// ---- DUTs/IO/Topology/Beckhoff_EJ5xxx_DF22D5A3.TcDUT
{attribute addProperty BoxType "EK1100-0000-0018"}
{attribute addProperty Id "Beckhoff_EJ5xxxEK1122Beckhoff_EJ5xxxEK1122_0744EC7C162A_0001_EJ5002_0000_0016EJ5002_8228306817822.25A_0002_EJ5002_0000_0017EJ5002_960CC6F117822.25A_0003_EJ5101_0000_0016EJ5101_6012872616220.25A_0004_EJ5151_0000_0016EJ5151_0AC1A36D19424.25"}
{attribute addProperty CRC "3743602083"}
{attribute addProperty SizeInBites "728"}
{attribute addProperty SizeInBytes "91"}
TYPE Beckhoff_EJ5xxx_DF22D5A3 EXTENDS EK1100_179A0949 :
STRUCT
	{attribute addProperty Name "Beckhoff_EJ5xxxEK1122"}
	Beckhoff_EJ5xxxEK1122 : Beckhoff_EJ5xxxEK1122_0744EC7C;
	{attribute addProperty Name "A_0001_EJ5002_0000_0016"}
	A_0001_EJ5002_0000_0016 : EJ5002_82283068;
	{attribute addProperty Name "A_0002_EJ5002_0000_0017"}
	A_0002_EJ5002_0000_0017 : EJ5002_960CC6F1;
	{attribute addProperty Name "A_0003_EJ5101_0000_0016"}
	A_0003_EJ5101_0000_0016 : EJ5101_60128726;
	{attribute addProperty Name "A_0004_EJ5151_0000_0016"}
	A_0004_EJ5151_0000_0016 : EJ5151_0AC1A36D;
END_STRUCT
END_TYPE

// ---- DUTs/IO/Topology/Beckhoff_EJ6xxxEK1122_30779985.TcDUT
{attribute addProperty BoxType "EK1122-0000-0018"}
{attribute addProperty Id "Beckhoff_EJ6xxxsub_EK1100EK1100_179A0949162"}
{attribute addProperty CRC "813144453"}
{attribute addProperty SizeInBites "16"}
{attribute addProperty SizeInBytes "2"}
TYPE Beckhoff_EJ6xxxEK1122_30779985 EXTENDS EK1122_179A0949 :
STRUCT
	{attribute addProperty Name "Beckhoff_EJ6xxxsub_EK1100"}
	Beckhoff_EJ6xxxsub_EK1100 : EK1100_179A0949;
END_STRUCT
END_TYPE

// ---- DUTs/IO/Topology/Beckhoff_EJ6xxx_A0E5C2C0.TcDUT
{attribute addProperty BoxType "EK1100-0000-0018"}
{attribute addProperty Id "Beckhoff_EJ6xxxEK1122Beckhoff_EJ6xxxEK1122_30779985162A_0001_EJ6002_0000_0016EJ6002_880A624E850106.25A_0002_EJ6224_0000_0016EJ6224_3990B4B417822.25A_0003_EJ6224_0090_0016EJ6224_3990B4B417822.25"}
{attribute addProperty CRC "2699412160"}
{attribute addProperty SizeInBites "1222"}
{attribute addProperty SizeInBytes "152.75"}
TYPE Beckhoff_EJ6xxx_A0E5C2C0 EXTENDS EK1100_179A0949 :
STRUCT
	{attribute addProperty Name "Beckhoff_EJ6xxxEK1122"}
	Beckhoff_EJ6xxxEK1122 : Beckhoff_EJ6xxxEK1122_30779985;
	{attribute addProperty Name "A_0001_EJ6002_0000_0016"}
	A_0001_EJ6002_0000_0016 : EJ6002_880A624E;
	{attribute addProperty Name "A_0002_EJ6224_0000_0016"}
	A_0002_EJ6224_0000_0016 : EJ6224_3990B4B4;
	{attribute addProperty Name "A_0003_EJ6224_0090_0016"}
	A_0003_EJ6224_0090_0016 : EJ6224_3990B4B4;
END_STRUCT
END_TYPE

// ---- DUTs/IO/Topology/Beckhoff_EJ7xxxEK1122_22994AD2.TcDUT
{attribute addProperty BoxType "EK1122-0000-0018"}
{attribute addProperty Id "Beckhoff_EJ7xxxsub_EK1100EK1100_179A0949162"}
{attribute addProperty CRC "580471506"}
{attribute addProperty SizeInBites "16"}
{attribute addProperty SizeInBytes "2"}
TYPE Beckhoff_EJ7xxxEK1122_22994AD2 EXTENDS EK1122_179A0949 :
STRUCT
	{attribute addProperty Name "Beckhoff_EJ7xxxsub_EK1100"}
	Beckhoff_EJ7xxxsub_EK1100 : EK1100_179A0949;
END_STRUCT
END_TYPE

// ---- DUTs/IO/Topology/Beckhoff_EJ7xxx_9F75012E.TcDUT
{attribute addProperty BoxType "EK1100-0000-0018"}
{attribute addProperty Id "Beckhoff_EJ7xxxEK1122Beckhoff_EJ7xxxEK1122_22994AD2162A_0001_EJ7031_0000_0026EJ7031_26D8313822628.25A_0002_EJ7037_0000_0020EJ7037_F30AD12822628.25A_0003_EJ7041_0052_0016EJ7041_26D8313822628.25A_0004_EJ7047_0000_0018EJ7047_F30AD12822628.25A_0005_EJ7047_0000_0019EJ7047_F30AD12822628.25A_0006_EJ7047_0000_0020EJ7047_F30AD12822628.25A_0007_EJ7342_0000_0019EJ7342_E03DC37137046.25A_0008_EJ7342_0000_0020EJ7342_E2585B8337046.25A_0009_EJ7211_0010_0026EJ7211_83D4128E25031.25A_0010_EJ7211_0010_0027EJ7211_83D4128E25031.25A_0011_EJ7211_0010_0028EJ7211_83D4128E25031.25A_0012_EJ7211_0010_0029EJ7211_83D4128E25031.25A_0013_EJ7211_0010_0030EJ7211_2D7B43DC25832.25A_0014_EJ7211_0010_0031EJ7211_2D7B43DC25832.25A_0015_EJ7211_0010_0032EJ7211_2D7B43DC25832.25A_0016_EJ7211_0011_0026EJ7211_789C0F5925031.25A_0017_EJ7211_0011_0027EJ7211_789C0F5925031.25A_0018_EJ7211_0011_0028EJ7211_789C0F5925031.25A_0019_EJ7211_0011_0029EJ7211_789C0F5925031.25A_0020_EJ7211_0011_0030EJ7211_789C0F5925031.25A_0021_EJ7211_0011_0031EJ7211_789C0F5925031.25A_0022_EJ7211_0011_0032EJ7211_789C0F5925031.25A_0023_EJ7211_9414_0029EJ7211_83D4128E25031.25A_0024_EJ7211_9414_0030EJ7211_5D87091826633.25A_0025_EJ7211_9414_0031EJ7211_5D87091826633.25A_0026_EJ7211_9414_0032EJ7211_5D87091826633.25A_0027_EJ7211_9415_0029EJ7211_789C0F5925031.25A_0028_EJ7211_9415_0030EJ7211_789C0F5925031.25A_0029_EJ7211_9415_0031EJ7211_789C0F5925031.25A_0030_EJ7211_9415_0032EJ7211_789C0F5925031.25A_0031_EJ7334_0008_0016EJ7334_68079CA927434.25A_0032_EJ7411_0000_0018EJ7411_675FBD0529036.25"}
{attribute addProperty CRC "2675245358"}
{attribute addProperty SizeInBites "8248"}
{attribute addProperty SizeInBytes "1031"}
TYPE Beckhoff_EJ7xxx_9F75012E EXTENDS EK1100_179A0949 :
STRUCT
	{attribute addProperty Name "Beckhoff_EJ7xxxEK1122"}
	Beckhoff_EJ7xxxEK1122 : Beckhoff_EJ7xxxEK1122_22994AD2;
	{attribute addProperty Name "A_0001_EJ7031_0000_0026"}
	A_0001_EJ7031_0000_0026 : EJ7031_26D83138;
	{attribute addProperty Name "A_0002_EJ7037_0000_0020"}
	A_0002_EJ7037_0000_0020 : EJ7037_F30AD128;
	{attribute addProperty Name "A_0003_EJ7041_0052_0016"}
	A_0003_EJ7041_0052_0016 : EJ7041_26D83138;
	{attribute addProperty Name "A_0004_EJ7047_0000_0018"}
	A_0004_EJ7047_0000_0018 : EJ7047_F30AD128;
	{attribute addProperty Name "A_0005_EJ7047_0000_0019"}
	A_0005_EJ7047_0000_0019 : EJ7047_F30AD128;
	{attribute addProperty Name "A_0006_EJ7047_0000_0020"}
	A_0006_EJ7047_0000_0020 : EJ7047_F30AD128;
	{attribute addProperty Name "A_0007_EJ7342_0000_0019"}
	A_0007_EJ7342_0000_0019 : EJ7342_E03DC371;
	{attribute addProperty Name "A_0008_EJ7342_0000_0020"}
	A_0008_EJ7342_0000_0020 : EJ7342_E2585B83;
	{attribute addProperty Name "A_0009_EJ7211_0010_0026"}
	A_0009_EJ7211_0010_0026 : EJ7211_83D4128E;
	{attribute addProperty Name "A_0010_EJ7211_0010_0027"}
	A_0010_EJ7211_0010_0027 : EJ7211_83D4128E;
	{attribute addProperty Name "A_0011_EJ7211_0010_0028"}
	A_0011_EJ7211_0010_0028 : EJ7211_83D4128E;
	{attribute addProperty Name "A_0012_EJ7211_0010_0029"}
	A_0012_EJ7211_0010_0029 : EJ7211_83D4128E;
	{attribute addProperty Name "A_0013_EJ7211_0010_0030"}
	A_0013_EJ7211_0010_0030 : EJ7211_2D7B43DC;
	{attribute addProperty Name "A_0014_EJ7211_0010_0031"}
	A_0014_EJ7211_0010_0031 : EJ7211_2D7B43DC;
	{attribute addProperty Name "A_0015_EJ7211_0010_0032"}
	A_0015_EJ7211_0010_0032 : EJ7211_2D7B43DC;
	{attribute addProperty Name "A_0016_EJ7211_0011_0026"}
	A_0016_EJ7211_0011_0026 : EJ7211_789C0F59;
	{attribute addProperty Name "A_0017_EJ7211_0011_0027"}
	A_0017_EJ7211_0011_0027 : EJ7211_789C0F59;
	{attribute addProperty Name "A_0018_EJ7211_0011_0028"}
	A_0018_EJ7211_0011_0028 : EJ7211_789C0F59;
	{attribute addProperty Name "A_0019_EJ7211_0011_0029"}
	A_0019_EJ7211_0011_0029 : EJ7211_789C0F59;
	{attribute addProperty Name "A_0020_EJ7211_0011_0030"}
	A_0020_EJ7211_0011_0030 : EJ7211_789C0F59;
	{attribute addProperty Name "A_0021_EJ7211_0011_0031"}
	A_0021_EJ7211_0011_0031 : EJ7211_789C0F59;
	{attribute addProperty Name "A_0022_EJ7211_0011_0032"}
	A_0022_EJ7211_0011_0032 : EJ7211_789C0F59;
	{attribute addProperty Name "A_0023_EJ7211_9414_0029"}
	A_0023_EJ7211_9414_0029 : EJ7211_83D4128E;
	{attribute addProperty Name "A_0024_EJ7211_9414_0030"}
	A_0024_EJ7211_9414_0030 : EJ7211_5D870918;
	{attribute addProperty Name "A_0025_EJ7211_9414_0031"}
	A_0025_EJ7211_9414_0031 : EJ7211_5D870918;
	{attribute addProperty Name "A_0026_EJ7211_9414_0032"}
	A_0026_EJ7211_9414_0032 : EJ7211_5D870918;
	{attribute addProperty Name "A_0027_EJ7211_9415_0029"}
	A_0027_EJ7211_9415_0029 : EJ7211_789C0F59;
	{attribute addProperty Name "A_0028_EJ7211_9415_0030"}
	A_0028_EJ7211_9415_0030 : EJ7211_789C0F59;
	{attribute addProperty Name "A_0029_EJ7211_9415_0031"}
	A_0029_EJ7211_9415_0031 : EJ7211_789C0F59;
	{attribute addProperty Name "A_0030_EJ7211_9415_0032"}
	A_0030_EJ7211_9415_0032 : EJ7211_789C0F59;
	{attribute addProperty Name "A_0031_EJ7334_0008_0016"}
	A_0031_EJ7334_0008_0016 : EJ7334_68079CA9;
	{attribute addProperty Name "A_0032_EJ7411_0000_0018"}
	A_0032_EJ7411_0000_0018 : EJ7411_675FBD05;
END_STRUCT
END_TYPE

// ---- DUTs/IO/Topology/Beckhoff_EJ9xxxEK1122_DB893B98.TcDUT
{attribute addProperty BoxType "EK1122-0000-0018"}
{attribute addProperty Id "Beckhoff_EJ9xxxsub_EK1100EK1100_179A0949162"}
{attribute addProperty CRC "3683203992"}
{attribute addProperty SizeInBites "16"}
{attribute addProperty SizeInBytes "2"}
TYPE Beckhoff_EJ9xxxEK1122_DB893B98 EXTENDS EK1122_179A0949 :
STRUCT
	{attribute addProperty Name "Beckhoff_EJ9xxxsub_EK1100"}
	Beckhoff_EJ9xxxsub_EK1100 : EK1100_179A0949;
END_STRUCT
END_TYPE

// ---- DUTs/IO/Topology/Beckhoff_EJ9xxx_660B2C8D.TcDUT
{attribute addProperty BoxType "EK1100-0000-0018"}
{attribute addProperty Id "Beckhoff_EJ9xxxEK1122Beckhoff_EJ9xxxEK1122_DB893B98162A_0001_EJ9001_0000_0016EJ9001_179A0949162A_0002_EJ9505_0000_0016EJ9505_13AAEB7E344.25A_0003_EJ9576_0000_0018EJ9576_30D5723B21026.25A_0004_EJ9576_0000_0019EJ9576_8602C5C421827.25A_0005_EJ9576_0000_0020EJ9576_EB67CEB421026.25A_0006_EJ9576_0000_0022EJ9576_EEF1625221827.25"}
{attribute addProperty CRC "1712008333"}
{attribute addProperty SizeInBites "922"}
{attribute addProperty SizeInBytes "115.25"}
TYPE Beckhoff_EJ9xxx_660B2C8D EXTENDS EK1100_179A0949 :
STRUCT
	{attribute addProperty Name "Beckhoff_EJ9xxxEK1122"}
	Beckhoff_EJ9xxxEK1122 : Beckhoff_EJ9xxxEK1122_DB893B98;
	{attribute addProperty Name "A_0001_EJ9001_0000_0016"}
	A_0001_EJ9001_0000_0016 : EJ9001_179A0949;
	{attribute addProperty Name "A_0002_EJ9505_0000_0016"}
	A_0002_EJ9505_0000_0016 : EJ9505_13AAEB7E;
	{attribute addProperty Name "A_0003_EJ9576_0000_0018"}
	A_0003_EJ9576_0000_0018 : EJ9576_30D5723B;
	{attribute addProperty Name "A_0004_EJ9576_0000_0019"}
	A_0004_EJ9576_0000_0019 : EJ9576_8602C5C4;
	{attribute addProperty Name "A_0005_EJ9576_0000_0020"}
	A_0005_EJ9576_0000_0020 : EJ9576_EB67CEB4;
	{attribute addProperty Name "A_0006_EJ9576_0000_0022"}
	A_0006_EJ9576_0000_0022 : EJ9576_EEF16252;
END_STRUCT
END_TYPE

// ---- DUTs/IO/Topology/Beckhoff_EJx9xxEK1122_05D2B413.TcDUT
{attribute addProperty BoxType "EK1122-0000-0018"}
{attribute addProperty Id "Beckhoff_EJx9xxsub_EK1100EK1100_179A0949162"}
{attribute addProperty CRC "97694739"}
{attribute addProperty SizeInBites "16"}
{attribute addProperty SizeInBytes "2"}
TYPE Beckhoff_EJx9xxEK1122_05D2B413 EXTENDS EK1122_179A0949 :
STRUCT
	{attribute addProperty Name "Beckhoff_EJx9xxsub_EK1100"}
	Beckhoff_EJx9xxsub_EK1100 : EK1100_179A0949;
END_STRUCT
END_TYPE

// ---- DUTs/IO/Topology/Beckhoff_EJx9xx_A9128509.TcDUT
{attribute addProperty BoxType "EK1100-0000-0018"}
{attribute addProperty Id "Beckhoff_EJx9xxEK1122Beckhoff_EJx9xxEK1122_05D2B413162A_0001_EJ1914_0000_0017EJ1914_5EB96E2D21026.25A_0002_EJ1914_0000_0018EJ1914_5EB96E2D21026.25A_0003_EJ1918_0000_0017EJ1918_151E5A8221827.25A_0004_EJ1918_0000_0018EJ1918_151E5A8221827.25A_0005_EJ1957_0000_0017EJ1957_6B6926D126032.5A_0006_EJ1957_0000_0018EJ1957_6B6926D126032.5A_0007_EJ2914_0000_0017EJ2914_46D107EB24430.5A_0008_EJ2914_0000_0018EJ2914_46D107EB24430.5A_0009_EJ2918_0000_0017EJ2918_AA36864B28435.5A_0010_EJ2918_0000_0018EJ2918_AA36864B28435.5A_0011_EJ6910_0000_0018EJ6910_4EA245C69812.25A_0012_EJ6910_0000_0020EJ6910_4EA245C69812.25"}
{attribute addProperty CRC "2836563209"}
{attribute addProperty SizeInBites "2644"}
{attribute addProperty SizeInBytes "330.5"}
TYPE Beckhoff_EJx9xx_A9128509 EXTENDS EK1100_179A0949 :
STRUCT
	{attribute addProperty Name "Beckhoff_EJx9xxEK1122"}
	Beckhoff_EJx9xxEK1122 : Beckhoff_EJx9xxEK1122_05D2B413;
	{attribute addProperty Name "A_0001_EJ1914_0000_0017"}
	A_0001_EJ1914_0000_0017 : EJ1914_5EB96E2D;
	{attribute addProperty Name "A_0002_EJ1914_0000_0018"}
	A_0002_EJ1914_0000_0018 : EJ1914_5EB96E2D;
	{attribute addProperty Name "A_0003_EJ1918_0000_0017"}
	A_0003_EJ1918_0000_0017 : EJ1918_151E5A82;
	{attribute addProperty Name "A_0004_EJ1918_0000_0018"}
	A_0004_EJ1918_0000_0018 : EJ1918_151E5A82;
	{attribute addProperty Name "A_0005_EJ1957_0000_0017"}
	A_0005_EJ1957_0000_0017 : EJ1957_6B6926D1;
	{attribute addProperty Name "A_0006_EJ1957_0000_0018"}
	A_0006_EJ1957_0000_0018 : EJ1957_6B6926D1;
	{attribute addProperty Name "A_0007_EJ2914_0000_0017"}
	A_0007_EJ2914_0000_0017 : EJ2914_46D107EB;
	{attribute addProperty Name "A_0008_EJ2914_0000_0018"}
	A_0008_EJ2914_0000_0018 : EJ2914_46D107EB;
	{attribute addProperty Name "A_0009_EJ2918_0000_0017"}
	A_0009_EJ2918_0000_0017 : EJ2918_AA36864B;
	{attribute addProperty Name "A_0010_EJ2918_0000_0018"}
	A_0010_EJ2918_0000_0018 : EJ2918_AA36864B;
	{attribute addProperty Name "A_0011_EJ6910_0000_0018"}
	A_0011_EJ6910_0000_0018 : EJ6910_4EA245C6;
	{attribute addProperty Name "A_0012_EJ6910_0000_0020"}
	A_0012_EJ6910_0000_0020 : EJ6910_4EA245C6;
END_STRUCT
END_TYPE

// ---- DUTs/IO/Topology/EtherCAT_Master_EJxxxx_24234FDA.TcDUT
{attribute addProperty BoxType "IODEVICETYPE_ETHERCATPROT"}
{attribute addProperty Id "Beckhoff_EJ1xxxBeckhoff_EJ1xxx_BA4DEDCC877109.625Beckhoff_EJ2xxxBeckhoff_EJ2xxx_42F4B05B1708213.5Beckhoff_EJ3xxxBeckhoff_EJ3xxx_F355313D4934616.75Beckhoff_EJ4xxxBeckhoff_EJ4xxx_B433EAC71353169.125Beckhoff_EJ5xxxBeckhoff_EJ5xxx_DF22D5A372891Beckhoff_EJ6xxxBeckhoff_EJ6xxx_A0E5C2C01222152.75Beckhoff_EJ7xxxBeckhoff_EJ7xxx_9F75012E82481031Beckhoff_EJ9xxxBeckhoff_EJ9xxx_660B2C8D922115.25Beckhoff_EJx9xxBeckhoff_EJx9xx_A91285092644330.5SyncUnitsSyncUnits_BBFB8ED413016.25InputsInputs_C3133F881088136OutputsOutputs_BAAAC74672090InfoDataInfoData_E9F65A829612"}
{attribute addProperty CRC "606293978"}
{attribute addProperty SizeInBites "24670"}
{attribute addProperty SizeInBytes "3083.75"}
TYPE EtherCAT_Master_EJxxxx_24234FDA :
STRUCT
	{attribute addProperty Name "Beckhoff_EJ1xxx"}
	Beckhoff_EJ1xxx : Beckhoff_EJ1xxx_BA4DEDCC;
	{attribute addProperty Name "Beckhoff_EJ2xxx"}
	Beckhoff_EJ2xxx : Beckhoff_EJ2xxx_42F4B05B;
	{attribute addProperty Name "Beckhoff_EJ3xxx"}
	Beckhoff_EJ3xxx : Beckhoff_EJ3xxx_F355313D;
	{attribute addProperty Name "Beckhoff_EJ4xxx"}
	Beckhoff_EJ4xxx : Beckhoff_EJ4xxx_B433EAC7;
	{attribute addProperty Name "Beckhoff_EJ5xxx"}
	Beckhoff_EJ5xxx : Beckhoff_EJ5xxx_DF22D5A3;
	{attribute addProperty Name "Beckhoff_EJ6xxx"}
	Beckhoff_EJ6xxx : Beckhoff_EJ6xxx_A0E5C2C0;
	{attribute addProperty Name "Beckhoff_EJ7xxx"}
	Beckhoff_EJ7xxx : Beckhoff_EJ7xxx_9F75012E;
	{attribute addProperty Name "Beckhoff_EJ9xxx"}
	Beckhoff_EJ9xxx : Beckhoff_EJ9xxx_660B2C8D;
	{attribute addProperty Name "Beckhoff_EJx9xx"}
	Beckhoff_EJx9xx : Beckhoff_EJx9xx_A9128509;
	{attribute addProperty Name "SyncUnits"}
	SyncUnits : SyncUnits_BBFB8ED4;
	{attribute addProperty Name "Inputs"}
	Inputs : Inputs_C3133F88;
	{attribute addProperty Name "Outputs"}
	Outputs : Outputs_BAAAC746;
	{attribute addProperty Name "InfoData"}
	InfoData : InfoData_E9F65A82;
END_STRUCT
END_TYPE

// ---- DUTs/IO/Topology/Beckhoff_EK11xxEK1122_0F9A1885.TcDUT
{attribute addProperty BoxType "EK1122-0000-0018"}
{attribute addProperty Id "Beckhoff_EK11xxsub_EK1100EK1100_179A0949162A_0001_EK1100_0000_0000EK1100_179A0949162A_0002_EK1100_0000_0001EK1100_179A0949162A_0003_EK1100_0000_0016EK1100_179A0949162A_0004_EK1100_0000_0017EK1100_179A0949162A_0005_EK1100_0000_0018EK1100_179A0949162A_0006_EK1100_0008_0016EK1100_179A0949162A_0009_EK1101_0000_0016EK1101_963BF4D7344.25A_0010_EK1101_0000_0017EK1101_963BF4D7344.25A_0011_EK1101_0000_0018EK1101_963BF4D7344.25A_0012_EK1101_0008_0016EK1101_963BF4D7344.25A_0013_EK1101_0010_0016EK1101_963BF4D7344.25A_0008_EK1100_0030_0017EK1100_179A0949162A_0007_EK1100_0030_0016EK1100_179A0949162"}
{attribute addProperty CRC "261757061"}
{attribute addProperty SizeInBites "314"}
{attribute addProperty SizeInBytes "39.25"}
TYPE Beckhoff_EK11xxEK1122_0F9A1885 EXTENDS EK1122_179A0949 :
STRUCT
	{attribute addProperty Name "Beckhoff_EK11xxsub_EK1100"}
	Beckhoff_EK11xxsub_EK1100 : EK1100_179A0949;
	{attribute addProperty Name "A_0001_EK1100_0000_0000"}
	A_0001_EK1100_0000_0000 : EK1100_179A0949;
	{attribute addProperty Name "A_0002_EK1100_0000_0001"}
	A_0002_EK1100_0000_0001 : EK1100_179A0949;
	{attribute addProperty Name "A_0003_EK1100_0000_0016"}
	A_0003_EK1100_0000_0016 : EK1100_179A0949;
	{attribute addProperty Name "A_0004_EK1100_0000_0017"}
	A_0004_EK1100_0000_0017 : EK1100_179A0949;
	{attribute addProperty Name "A_0005_EK1100_0000_0018"}
	A_0005_EK1100_0000_0018 : EK1100_179A0949;
	{attribute addProperty Name "A_0006_EK1100_0008_0016"}
	A_0006_EK1100_0008_0016 : EK1100_179A0949;
	{attribute addProperty Name "A_0009_EK1101_0000_0016"}
	A_0009_EK1101_0000_0016 : EK1101_963BF4D7;
	{attribute addProperty Name "A_0010_EK1101_0000_0017"}
	A_0010_EK1101_0000_0017 : EK1101_963BF4D7;
	{attribute addProperty Name "A_0011_EK1101_0000_0018"}
	A_0011_EK1101_0000_0018 : EK1101_963BF4D7;
	{attribute addProperty Name "A_0012_EK1101_0008_0016"}
	A_0012_EK1101_0008_0016 : EK1101_963BF4D7;
	{attribute addProperty Name "A_0013_EK1101_0010_0016"}
	A_0013_EK1101_0010_0016 : EK1101_963BF4D7;
	{attribute addProperty Name "A_0008_EK1100_0030_0017"}
	A_0008_EK1100_0030_0017 : EK1100_179A0949;
	{attribute addProperty Name "A_0007_EK1100_0030_0016"}
	A_0007_EK1100_0030_0016 : EK1100_179A0949;
END_STRUCT
END_TYPE

// ---- DUTs/IO/Topology/Beckhoff_EK11xx_C12453FF.TcDUT
{attribute addProperty BoxType "EK1100-0000-0018"}
{attribute addProperty Id "Beckhoff_EK11xxEK1122Beckhoff_EK11xxEK1122_0F9A188531439.25A_0018_EK1110_0043_0016EK1110_179A0949162A_0024_EK1122_0008_0016EK1122_179A0949162A_0023_EK1122_0000_0018EK1122_179A0949162A_0022_EK1122_0000_0017EK1122_179A0949162A_0021_EK1122_0000_0016EK1122_179A0949162A_0020_EK1121_0010_0016EK1121_179A0949162A_0019_EK1110_0044_0016EK1110_179A0949162A_0017_EK1110_0008_0016EK1110_179A0949162A_0016_EK1110_0000_0017EK1110_179A0949162A_0015_EK1110_0000_0016EK1110_179A0949162A_0014_EK1110_0000_0000EK1110_179A0949162"}
{attribute addProperty CRC "3240383487"}
{attribute addProperty SizeInBites "490"}
{attribute addProperty SizeInBytes "61.25"}
TYPE Beckhoff_EK11xx_C12453FF EXTENDS EK1100_179A0949 :
STRUCT
	{attribute addProperty Name "Beckhoff_EK11xxEK1122"}
	Beckhoff_EK11xxEK1122 : Beckhoff_EK11xxEK1122_0F9A1885;
	{attribute addProperty Name "A_0018_EK1110_0043_0016"}
	A_0018_EK1110_0043_0016 : EK1110_179A0949;
	{attribute addProperty Name "A_0024_EK1122_0008_0016"}
	A_0024_EK1122_0008_0016 : EK1122_179A0949;
	{attribute addProperty Name "A_0023_EK1122_0000_0018"}
	A_0023_EK1122_0000_0018 : EK1122_179A0949;
	{attribute addProperty Name "A_0022_EK1122_0000_0017"}
	A_0022_EK1122_0000_0017 : EK1122_179A0949;
	{attribute addProperty Name "A_0021_EK1122_0000_0016"}
	A_0021_EK1122_0000_0016 : EK1122_179A0949;
	{attribute addProperty Name "A_0020_EK1121_0010_0016"}
	A_0020_EK1121_0010_0016 : EK1121_179A0949;
	{attribute addProperty Name "A_0019_EK1110_0044_0016"}
	A_0019_EK1110_0044_0016 : EK1110_179A0949;
	{attribute addProperty Name "A_0017_EK1110_0008_0016"}
	A_0017_EK1110_0008_0016 : EK1110_179A0949;
	{attribute addProperty Name "A_0016_EK1110_0000_0017"}
	A_0016_EK1110_0000_0017 : EK1110_179A0949;
	{attribute addProperty Name "A_0015_EK1110_0000_0016"}
	A_0015_EK1110_0000_0016 : EK1110_179A0949;
	{attribute addProperty Name "A_0014_EK1110_0000_0000"}
	A_0014_EK1110_0000_0000 : EK1110_179A0949;
END_STRUCT
END_TYPE

// ---- DUTs/IO/Topology/Beckhoff_EK12xxEK1122_E9998301.TcDUT
{attribute addProperty BoxType "EK1122-0000-0018"}
{attribute addProperty Id "Beckhoff_EK12xxsub_EK1100EK1100_179A0949162"}
{attribute addProperty CRC "3919151873"}
{attribute addProperty SizeInBites "16"}
{attribute addProperty SizeInBytes "2"}
TYPE Beckhoff_EK12xxEK1122_E9998301 EXTENDS EK1122_179A0949 :
STRUCT
	{attribute addProperty Name "Beckhoff_EK12xxsub_EK1100"}
	Beckhoff_EK12xxsub_EK1100 : EK1100_179A0949;
END_STRUCT
END_TYPE

// ---- DUTs/IO/Topology/Beckhoff_EK12xx_26FD3E4A.TcDUT
{attribute addProperty BoxType "EK1100-0000-0018"}
{attribute addProperty Id "Beckhoff_EK12xxEK1122Beckhoff_EK12xxEK1122_E9998301162"}
{attribute addProperty CRC "654130762"}
{attribute addProperty SizeInBites "16"}
{attribute addProperty SizeInBytes "2"}
TYPE Beckhoff_EK12xx_26FD3E4A EXTENDS EK1100_179A0949 :
STRUCT
	{attribute addProperty Name "Beckhoff_EK12xxEK1122"}
	Beckhoff_EK12xxEK1122 : Beckhoff_EK12xxEK1122_E9998301;
END_STRUCT
END_TYPE

// ---- DUTs/IO/Topology/Beckhoff_EK13xxEK1122_7883D180.TcDUT
{attribute addProperty BoxType "EK1122-0000-0018"}
{attribute addProperty Id "Beckhoff_EK13xxsub_EK1100EK1100_179A0949162A_0001_EK1300_0000_0017EK1300_0EEAC8F2344.25"}
{attribute addProperty CRC "2021904768"}
{attribute addProperty SizeInBites "50"}
{attribute addProperty SizeInBytes "6.25"}
TYPE Beckhoff_EK13xxEK1122_7883D180 EXTENDS EK1122_179A0949 :
STRUCT
	{attribute addProperty Name "Beckhoff_EK13xxsub_EK1100"}
	Beckhoff_EK13xxsub_EK1100 : EK1100_179A0949;
	{attribute addProperty Name "A_0001_EK1300_0000_0017"}
	A_0001_EK1300_0000_0017 : EK1300_0EEAC8F2;
END_STRUCT
END_TYPE

// ---- DUTs/IO/Topology/Beckhoff_EK13xx_F78FC0F8.TcDUT
{attribute addProperty BoxType "EK1100-0000-0018"}
{attribute addProperty Id "Beckhoff_EK13xxEK1122Beckhoff_EK13xxEK1122_7883D180506.25A_0003_EK1322_0000_0017EK1322_0EEAC8F2344.25A_0002_EK1310_0000_0017EK1310_0EEAC8F2344.25"}
{attribute addProperty CRC "4153393400"}
{attribute addProperty SizeInBites "118"}
{attribute addProperty SizeInBytes "14.75"}
TYPE Beckhoff_EK13xx_F78FC0F8 EXTENDS EK1100_179A0949 :
STRUCT
	{attribute addProperty Name "Beckhoff_EK13xxEK1122"}
	Beckhoff_EK13xxEK1122 : Beckhoff_EK13xxEK1122_7883D180;
	{attribute addProperty Name "A_0003_EK1322_0000_0017"}
	A_0003_EK1322_0000_0017 : EK1322_0EEAC8F2;
	{attribute addProperty Name "A_0002_EK1310_0000_0017"}
	A_0002_EK1310_0000_0017 : EK1310_0EEAC8F2;
END_STRUCT
END_TYPE

// ---- DUTs/IO/Topology/Beckhoff_EK15xxEK1122_F4825052.TcDUT
{attribute addProperty BoxType "EK1122-0000-0018"}
{attribute addProperty Id "Beckhoff_EK15xxsub_EK1100EK1100_179A0949162A_0001_EK1501_0000_0016EK1501_963BF4D7344.25A_0002_EK1501_0000_0017EK1501_963BF4D7344.25A_0003_EK1501_0000_0018EK1501_963BF4D7344.25A_0004_EK1501_0000_0019EK1501_963BF4D7344.25A_0005_EK1501_0010_0016EK1501_963BF4D7344.25A_0006_EK1501_0010_0017EK1501_963BF4D7344.25A_0007_EK1501_0010_0018EK1501_963BF4D7344.25A_0008_EK1501_0100_0016EK1501_963BF4D7344.25A_0020_EK1541_0000_0016EK1541_963BF4D7344.25A_0021_EK1541_0000_0017EK1541_963BF4D7344.25A_0022_EK1541_0000_0018EK1541_963BF4D7344.25"}
{attribute addProperty CRC "4102180946"}
{attribute addProperty SizeInBites "390"}
{attribute addProperty SizeInBytes "48.75"}
TYPE Beckhoff_EK15xxEK1122_F4825052 EXTENDS EK1122_179A0949 :
STRUCT
	{attribute addProperty Name "Beckhoff_EK15xxsub_EK1100"}
	Beckhoff_EK15xxsub_EK1100 : EK1100_179A0949;
	{attribute addProperty Name "A_0001_EK1501_0000_0016"}
	A_0001_EK1501_0000_0016 : EK1501_963BF4D7;
	{attribute addProperty Name "A_0002_EK1501_0000_0017"}
	A_0002_EK1501_0000_0017 : EK1501_963BF4D7;
	{attribute addProperty Name "A_0003_EK1501_0000_0018"}
	A_0003_EK1501_0000_0018 : EK1501_963BF4D7;
	{attribute addProperty Name "A_0004_EK1501_0000_0019"}
	A_0004_EK1501_0000_0019 : EK1501_963BF4D7;
	{attribute addProperty Name "A_0005_EK1501_0010_0016"}
	A_0005_EK1501_0010_0016 : EK1501_963BF4D7;
	{attribute addProperty Name "A_0006_EK1501_0010_0017"}
	A_0006_EK1501_0010_0017 : EK1501_963BF4D7;
	{attribute addProperty Name "A_0007_EK1501_0010_0018"}
	A_0007_EK1501_0010_0018 : EK1501_963BF4D7;
	{attribute addProperty Name "A_0008_EK1501_0100_0016"}
	A_0008_EK1501_0100_0016 : EK1501_963BF4D7;
	{attribute addProperty Name "A_0020_EK1541_0000_0016"}
	A_0020_EK1541_0000_0016 : EK1541_963BF4D7;
	{attribute addProperty Name "A_0021_EK1541_0000_0017"}
	A_0021_EK1541_0000_0017 : EK1541_963BF4D7;
	{attribute addProperty Name "A_0022_EK1541_0000_0018"}
	A_0022_EK1541_0000_0018 : EK1541_963BF4D7;
END_STRUCT
END_TYPE

// ---- DUTs/IO/Topology/Beckhoff_EK15xx_2CCE234B.TcDUT
{attribute addProperty BoxType "EK1100-0000-0018"}
{attribute addProperty Id "Beckhoff_EK15xxEK1122Beckhoff_EK15xxEK1122_F482505239048.75A_0025_EK1561_0000_0018EK1561_179A0949162A_0024_EK1561_0000_0017EK1561_179A0949162A_0023_EK1561_0000_0016EK1561_179A0949162A_0019_EK1521_0010_0020EK1521_179A0949162A_0018_EK1521_0010_0019EK1521_179A0949162A_0017_EK1521_0010_0018EK1521_179A0949162A_0016_EK1521_0010_0017EK1521_179A0949162A_0015_EK1521_0010_0016EK1521_179A0949162A_0014_EK1521_0000_0021EK1521_179A0949162A_0013_EK1521_0000_0020EK1521_179A0949162A_0012_EK1521_0000_0019EK1521_179A0949162A_0011_EK1521_0000_0018EK1521_179A0949162A_0010_EK1521_0000_0017EK1521_179A0949162A_0009_EK1521_0000_0016EK1521_179A0949162"}
{attribute addProperty CRC "751706955"}
{attribute addProperty SizeInBites "614"}
{attribute addProperty SizeInBytes "76.75"}
TYPE Beckhoff_EK15xx_2CCE234B EXTENDS EK1100_179A0949 :
STRUCT
	{attribute addProperty Name "Beckhoff_EK15xxEK1122"}
	Beckhoff_EK15xxEK1122 : Beckhoff_EK15xxEK1122_F4825052;
	{attribute addProperty Name "A_0025_EK1561_0000_0018"}
	A_0025_EK1561_0000_0018 : EK1561_179A0949;
	{attribute addProperty Name "A_0024_EK1561_0000_0017"}
	A_0024_EK1561_0000_0017 : EK1561_179A0949;
	{attribute addProperty Name "A_0023_EK1561_0000_0016"}
	A_0023_EK1561_0000_0016 : EK1561_179A0949;
	{attribute addProperty Name "A_0019_EK1521_0010_0020"}
	A_0019_EK1521_0010_0020 : EK1521_179A0949;
	{attribute addProperty Name "A_0018_EK1521_0010_0019"}
	A_0018_EK1521_0010_0019 : EK1521_179A0949;
	{attribute addProperty Name "A_0017_EK1521_0010_0018"}
	A_0017_EK1521_0010_0018 : EK1521_179A0949;
	{attribute addProperty Name "A_0016_EK1521_0010_0017"}
	A_0016_EK1521_0010_0017 : EK1521_179A0949;
	{attribute addProperty Name "A_0015_EK1521_0010_0016"}
	A_0015_EK1521_0010_0016 : EK1521_179A0949;
	{attribute addProperty Name "A_0014_EK1521_0000_0021"}
	A_0014_EK1521_0000_0021 : EK1521_179A0949;
	{attribute addProperty Name "A_0013_EK1521_0000_0020"}
	A_0013_EK1521_0000_0020 : EK1521_179A0949;
	{attribute addProperty Name "A_0012_EK1521_0000_0019"}
	A_0012_EK1521_0000_0019 : EK1521_179A0949;
	{attribute addProperty Name "A_0011_EK1521_0000_0018"}
	A_0011_EK1521_0000_0018 : EK1521_179A0949;
	{attribute addProperty Name "A_0010_EK1521_0000_0017"}
	A_0010_EK1521_0000_0017 : EK1521_179A0949;
	{attribute addProperty Name "A_0009_EK1521_0000_0016"}
	A_0009_EK1521_0000_0016 : EK1521_179A0949;
END_STRUCT
END_TYPE

// ---- DUTs/IO/Topology/Beckhoff_EK18xxEK1122_46BB19D8.TcDUT
{attribute addProperty BoxType "EK1122-0000-0018"}
{attribute addProperty Id "Beckhoff_EK18xxsub_EK1100EK1100_179A0949162A_0001_EK1814_0000_0016EK1814_97B4DD118210.25A_0002_EK1814_0000_0017EK1814_97B4DD118210.25A_0003_EK1814_0000_0018EK1814_97B4DD118210.25A_0004_EK1814_0000_0019EK1814_97B4DD118210.25A_0005_EK1818_0000_0016EK1818_5F755A8411414.25A_0006_EK1818_0000_0017EK1818_5F755A8411414.25A_0007_EK1818_0000_0018EK1818_5F755A8411414.25A_0008_EK1828_0000_0016EK1828_A5978B6311414.25A_0009_EK1828_0000_0017EK1828_A5978B6311414.25A_0010_EK1828_0000_0018EK1828_A5978B6311414.25A_0011_EK1828_0010_0016EK1828_A854BE6D8110.125A_0012_EK1828_0010_0017EK1828_A854BE6D8110.125A_0013_EK1828_0010_0018EK1828_A854BE6D8110.125"}
{attribute addProperty CRC "1186666968"}
{attribute addProperty SizeInBites "1271"}
{attribute addProperty SizeInBytes "158.875"}
TYPE Beckhoff_EK18xxEK1122_46BB19D8 EXTENDS EK1122_179A0949 :
STRUCT
	{attribute addProperty Name "Beckhoff_EK18xxsub_EK1100"}
	Beckhoff_EK18xxsub_EK1100 : EK1100_179A0949;
	{attribute addProperty Name "A_0001_EK1814_0000_0016"}
	A_0001_EK1814_0000_0016 : EK1814_97B4DD11;
	{attribute addProperty Name "A_0002_EK1814_0000_0017"}
	A_0002_EK1814_0000_0017 : EK1814_97B4DD11;
	{attribute addProperty Name "A_0003_EK1814_0000_0018"}
	A_0003_EK1814_0000_0018 : EK1814_97B4DD11;
	{attribute addProperty Name "A_0004_EK1814_0000_0019"}
	A_0004_EK1814_0000_0019 : EK1814_97B4DD11;
	{attribute addProperty Name "A_0005_EK1818_0000_0016"}
	A_0005_EK1818_0000_0016 : EK1818_5F755A84;
	{attribute addProperty Name "A_0006_EK1818_0000_0017"}
	A_0006_EK1818_0000_0017 : EK1818_5F755A84;
	{attribute addProperty Name "A_0007_EK1818_0000_0018"}
	A_0007_EK1818_0000_0018 : EK1818_5F755A84;
	{attribute addProperty Name "A_0008_EK1828_0000_0016"}
	A_0008_EK1828_0000_0016 : EK1828_A5978B63;
	{attribute addProperty Name "A_0009_EK1828_0000_0017"}
	A_0009_EK1828_0000_0017 : EK1828_A5978B63;
	{attribute addProperty Name "A_0010_EK1828_0000_0018"}
	A_0010_EK1828_0000_0018 : EK1828_A5978B63;
	{attribute addProperty Name "A_0011_EK1828_0010_0016"}
	A_0011_EK1828_0010_0016 : EK1828_A854BE6D;
	{attribute addProperty Name "A_0012_EK1828_0010_0017"}
	A_0012_EK1828_0010_0017 : EK1828_A854BE6D;
	{attribute addProperty Name "A_0013_EK1828_0010_0018"}
	A_0013_EK1828_0010_0018 : EK1828_A854BE6D;
END_STRUCT
END_TYPE

// ---- DUTs/IO/Topology/Beckhoff_EK18xx_2BB31392.TcDUT
{attribute addProperty BoxType "EK1100-0000-0018"}
{attribute addProperty Id "Beckhoff_EK18xxEK1122Beckhoff_EK18xxEK1122_46BB19D81271158.875"}
{attribute addProperty CRC "733156242"}
{attribute addProperty SizeInBites "1271"}
{attribute addProperty SizeInBytes "158.875"}
TYPE Beckhoff_EK18xx_2BB31392 EXTENDS EK1100_179A0949 :
STRUCT
	{attribute addProperty Name "Beckhoff_EK18xxEK1122"}
	Beckhoff_EK18xxEK1122 : Beckhoff_EK18xxEK1122_46BB19D8;
END_STRUCT
END_TYPE

// ---- DUTs/IO/Topology/Beckhoff_EKM1xxxEK1122_7DC4CCD1.TcDUT
{attribute addProperty BoxType "EK1122-0000-0018"}
{attribute addProperty Id "Beckhoff_EKM1xxxsub_EK1100EK1100_179A0949162A_0001_EKM1101_0000_0016EKM1101_87969BFD51464.25A_0002_EKM1101_0000_0017EKM1101_87969BFD51464.25A_0003_EKM1101_0000_0018EKM1101_87969BFD51464.25A_0004_EKM1101_0000_0019EKM1101_87969BFD51464.25A_0005_EKM1101_0000_0020EKM1101_87969BFD51464.25"}
{attribute addProperty CRC "2110049489"}
{attribute addProperty SizeInBites "2586"}
{attribute addProperty SizeInBytes "323.25"}
TYPE Beckhoff_EKM1xxxEK1122_7DC4CCD1 EXTENDS EK1122_179A0949 :
STRUCT
	{attribute addProperty Name "Beckhoff_EKM1xxxsub_EK1100"}
	Beckhoff_EKM1xxxsub_EK1100 : EK1100_179A0949;
	{attribute addProperty Name "A_0001_EKM1101_0000_0016"}
	A_0001_EKM1101_0000_0016 : EKM1101_87969BFD;
	{attribute addProperty Name "A_0002_EKM1101_0000_0017"}
	A_0002_EKM1101_0000_0017 : EKM1101_87969BFD;
	{attribute addProperty Name "A_0003_EKM1101_0000_0018"}
	A_0003_EKM1101_0000_0018 : EKM1101_87969BFD;
	{attribute addProperty Name "A_0004_EKM1101_0000_0019"}
	A_0004_EKM1101_0000_0019 : EKM1101_87969BFD;
	{attribute addProperty Name "A_0005_EKM1101_0000_0020"}
	A_0005_EKM1101_0000_0020 : EKM1101_87969BFD;
END_STRUCT
END_TYPE

// ---- DUTs/IO/Topology/Beckhoff_EKM1xxx_A6D53207.TcDUT
{attribute addProperty BoxType "EK1100-0000-0018"}
{attribute addProperty Id "Beckhoff_EKM1xxxEK1122Beckhoff_EKM1xxxEK1122_7DC4CCD12586323.25"}
{attribute addProperty CRC "2798989831"}
{attribute addProperty SizeInBites "2586"}
{attribute addProperty SizeInBytes "323.25"}
TYPE Beckhoff_EKM1xxx_A6D53207 EXTENDS EK1100_179A0949 :
STRUCT
	{attribute addProperty Name "Beckhoff_EKM1xxxEK1122"}
	Beckhoff_EKM1xxxEK1122 : Beckhoff_EKM1xxxEK1122_7DC4CCD1;
END_STRUCT
END_TYPE

// ---- DUTs/IO/Topology/Beckhoff_EKx9xxEK1122_199990A5.TcDUT
{attribute addProperty BoxType "EK1122-0000-0018"}
{attribute addProperty Id "Beckhoff_EKx9xxsub_EK1100EK1100_179A0949162A_0001_EK1960_0000_0019EK1960_D284ECC656470.5A_0002_EK1960_0000_0021EK1960_858568AC53266.5A_0003_EK1960_0008_0019EK1960_D284ECC656470.5A_0004_EK1960_0008_0021EK1960_858568AC53266.5A_0005_EK1960_2600_0019EK1960_48A2E24356470.5A_0006_EK1960_2600_0021EK1960_3617E9AF56470.5A_0007_EK1960_2608_0019EK1960_48A2E24356470.5A_0008_EK1960_2608_0021EK1960_3617E9AF56470.5"}
{attribute addProperty CRC "429494437"}
{attribute addProperty SizeInBites "4464"}
{attribute addProperty SizeInBytes "558"}
TYPE Beckhoff_EKx9xxEK1122_199990A5 EXTENDS EK1122_179A0949 :
STRUCT
	{attribute addProperty Name "Beckhoff_EKx9xxsub_EK1100"}
	Beckhoff_EKx9xxsub_EK1100 : EK1100_179A0949;
	{attribute addProperty Name "A_0001_EK1960_0000_0019"}
	A_0001_EK1960_0000_0019 : EK1960_D284ECC6;
	{attribute addProperty Name "A_0002_EK1960_0000_0021"}
	A_0002_EK1960_0000_0021 : EK1960_858568AC;
	{attribute addProperty Name "A_0003_EK1960_0008_0019"}
	A_0003_EK1960_0008_0019 : EK1960_D284ECC6;
	{attribute addProperty Name "A_0004_EK1960_0008_0021"}
	A_0004_EK1960_0008_0021 : EK1960_858568AC;
	{attribute addProperty Name "A_0005_EK1960_2600_0019"}
	A_0005_EK1960_2600_0019 : EK1960_48A2E243;
	{attribute addProperty Name "A_0006_EK1960_2600_0021"}
	A_0006_EK1960_2600_0021 : EK1960_3617E9AF;
	{attribute addProperty Name "A_0007_EK1960_2608_0019"}
	A_0007_EK1960_2608_0019 : EK1960_48A2E243;
	{attribute addProperty Name "A_0008_EK1960_2608_0021"}
	A_0008_EK1960_2608_0021 : EK1960_3617E9AF;
END_STRUCT
END_TYPE

// ---- DUTs/IO/Topology/Beckhoff_EKx9xx_14304971.TcDUT
{attribute addProperty BoxType "EK1100-0000-0018"}
{attribute addProperty Id "Beckhoff_EKx9xxEK1122Beckhoff_EKx9xxEK1122_199990A54464558"}
{attribute addProperty CRC "338708849"}
{attribute addProperty SizeInBites "4464"}
{attribute addProperty SizeInBytes "558"}
TYPE Beckhoff_EKx9xx_14304971 EXTENDS EK1100_179A0949 :
STRUCT
	{attribute addProperty Name "Beckhoff_EKx9xxEK1122"}
	Beckhoff_EKx9xxEK1122 : Beckhoff_EKx9xxEK1122_199990A5;
END_STRUCT
END_TYPE

// ---- DUTs/IO/Topology/Beckhoff_EKxxxx_0080EK1122_49C116CC.TcDUT
{attribute addProperty BoxType "EK1122-0000-0018"}
{attribute addProperty Id "Beckhoff_EKxxxx_0080sub_EK1100EK1100_179A0949162"}
{attribute addProperty CRC "1237391052"}
{attribute addProperty SizeInBites "16"}
{attribute addProperty SizeInBytes "2"}
TYPE Beckhoff_EKxxxx_0080EK1122_49C116CC EXTENDS EK1122_179A0949 :
STRUCT
	{attribute addProperty Name "Beckhoff_EKxxxx_0080sub_EK1100"}
	Beckhoff_EKxxxx_0080sub_EK1100 : EK1100_179A0949;
END_STRUCT
END_TYPE

// ---- DUTs/IO/Topology/Beckhoff_EKxxxx_0080_F8E2E0BC.TcDUT
{attribute addProperty BoxType "EK1100-0000-0018"}
{attribute addProperty Id "Beckhoff_EKxxxx_0080EK1122Beckhoff_EKxxxx_0080EK1122_49C116CC162A_0006_EK1122_0080_0019EK1122_179A0949162A_0005_EK1122_0080_0018EK1122_179A0949162A_0004_EK1122_0080_0017EK1122_179A0949162"}
{attribute addProperty CRC "4175618236"}
{attribute addProperty SizeInBites "64"}
{attribute addProperty SizeInBytes "8"}
TYPE Beckhoff_EKxxxx_0080_F8E2E0BC EXTENDS EK1100_179A0949 :
STRUCT
	{attribute addProperty Name "Beckhoff_EKxxxx_0080EK1122"}
	Beckhoff_EKxxxx_0080EK1122 : Beckhoff_EKxxxx_0080EK1122_49C116CC;
	{attribute addProperty Name "A_0006_EK1122_0080_0019"}
	A_0006_EK1122_0080_0019 : EK1122_179A0949;
	{attribute addProperty Name "A_0005_EK1122_0080_0018"}
	A_0005_EK1122_0080_0018 : EK1122_179A0949;
	{attribute addProperty Name "A_0004_EK1122_0080_0017"}
	A_0004_EK1122_0080_0017 : EK1122_179A0949;
END_STRUCT
END_TYPE

// ---- DUTs/IO/Topology/EtherCAT_Master_EKxxxx_0AF69055.TcDUT
{attribute addProperty BoxType "IODEVICETYPE_ETHERCATPROT"}
{attribute addProperty Id "Beckhoff_EK11xxBeckhoff_EK11xx_C12453FF49061.25Beckhoff_EK12xxBeckhoff_EK12xx_26FD3E4A162Beckhoff_EK13xxBeckhoff_EK13xx_F78FC0F811814.75Beckhoff_EK15xxBeckhoff_EK15xx_2CCE234B61476.75Beckhoff_EK18xxBeckhoff_EK18xx_2BB313921271158.875Beckhoff_EKM1xxxBeckhoff_EKM1xxx_A6D532072586323.25Beckhoff_EKx9xxBeckhoff_EKx9xx_143049714464558Beckhoff_EKxxxx_0080Beckhoff_EKxxxx_0080_F8E2E0BC648SyncUnitsSyncUnits_BBFB8ED413016.25InputsInputs_C3133F881088136OutputsOutputs_BAAAC74672090InfoDataInfoData_E9F65A829612"}
{attribute addProperty CRC "183930965"}
{attribute addProperty SizeInBites "11657"}
{attribute addProperty SizeInBytes "1457.125"}
TYPE EtherCAT_Master_EKxxxx_0AF69055 :
STRUCT
	{attribute addProperty Name "Beckhoff_EK11xx"}
	Beckhoff_EK11xx : Beckhoff_EK11xx_C12453FF;
	{attribute addProperty Name "Beckhoff_EK12xx"}
	Beckhoff_EK12xx : Beckhoff_EK12xx_26FD3E4A;
	{attribute addProperty Name "Beckhoff_EK13xx"}
	Beckhoff_EK13xx : Beckhoff_EK13xx_F78FC0F8;
	{attribute addProperty Name "Beckhoff_EK15xx"}
	Beckhoff_EK15xx : Beckhoff_EK15xx_2CCE234B;
	{attribute addProperty Name "Beckhoff_EK18xx"}
	Beckhoff_EK18xx : Beckhoff_EK18xx_2BB31392;
	{attribute addProperty Name "Beckhoff_EKM1xxx"}
	Beckhoff_EKM1xxx : Beckhoff_EKM1xxx_A6D53207;
	{attribute addProperty Name "Beckhoff_EKx9xx"}
	Beckhoff_EKx9xx : Beckhoff_EKx9xx_14304971;
	{attribute addProperty Name "Beckhoff_EKxxxx_0080"}
	Beckhoff_EKxxxx_0080 : Beckhoff_EKxxxx_0080_F8E2E0BC;
	{attribute addProperty Name "SyncUnits"}
	SyncUnits : SyncUnits_BBFB8ED4;
	{attribute addProperty Name "Inputs"}
	Inputs : Inputs_C3133F88;
	{attribute addProperty Name "Outputs"}
	Outputs : Outputs_BAAAC746;
	{attribute addProperty Name "InfoData"}
	InfoData : InfoData_E9F65A82;
END_STRUCT
END_TYPE

// ---- GVLs/GVL_iXlinker.TcGVL
{attribute 'qualified_only'}
VAR_GLOBAL
		EtherCAT_Master_EJxxxx : EtherCAT_Master_EJxxxx_24234FDA;
		EtherCAT_Master_EKxxxx : EtherCAT_Master_EKxxxx_0AF69055;
END_VAR
